PROGRAM MAIN
VAR
	fbReadCoilExample : FB_ReadCoilExample;
END_VAR

fbReadCoilExample();

END_PROGRAM

(* stored: Version 1.1.0.1, ProductVersion 3.1.4024.12
   POU MAIN: Id {28c255d8-6965-4217-82e9-a941df42268f}, SpecialFunc None *)
